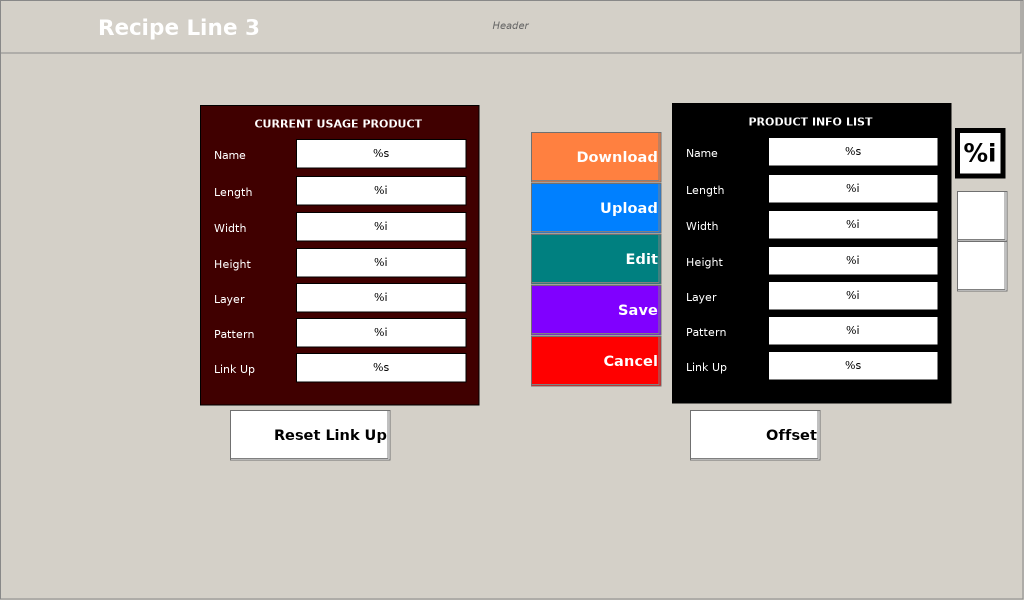
VISUALIZATION MRecipe_3  // 1024x600
    Frame (0,-2 1021x55)
        shows Header()
    Label (95,15 250x25), "Recipe Line 3"
    RoundedRectangle (672,103 279x300)
    Label (697,102 227x40), "PRODUCT INFO LIST"
    Label (683,136 78x35), "Name"
    RoundedRectangle (768,137 170x29), "%s", text variable: HMI_GVL.arRecipeHMI[3].ProductName, input disabled if: Status_GVL.StsEdit[3]
        OnMouseClick: write the text variable via Default
    Label (683,173 78x35), "Length"
    RoundedRectangle (768,174 170x29), "%i", text variable: HMI_GVL.arRecipeHMI[3].ProductLength, input disabled if: Status_GVL.StsEdit[3]
        OnMouseClick: write the text variable via Default
    Label (683,209 78x35), "Width"
    RoundedRectangle (768,210 170x29), "%i", text variable: HMI_GVL.arRecipeHMI[3].ProductWidth, input disabled if: Status_GVL.StsEdit[3]
        OnMouseClick: write the text variable via Default
    Label (683,245 78x35), "Height"
    RoundedRectangle (768,246 170x29), "%i", text variable: HMI_GVL.arRecipeHMI[3].ProductHeight, input disabled if: Status_GVL.StsEdit[3]
        OnMouseClick: write the text variable via Default
    Label (683,280 78x35), "Layer"
    RoundedRectangle (768,281 170x29), "%i", text variable: HMI_GVL.arRecipeHMI[3].Stacking, input disabled if: Status_GVL.StsEdit[3]
        OnMouseClick: write the text variable via Default
    Label (683,315 78x35), "Pattern"
    RoundedRectangle (768,316 170x29), "%i", text variable: HMI_GVL.arRecipeHMI[3].ProductPattern, input disabled if: Status_GVL.StsEdit[3]
        OnMouseClick: write the text variable via Default
    Label (683,350 78x35), "Link Up"
    RoundedRectangle (768,351 170x29), "%s", text variable: HMI_GVL.arRecipeHMI[3].LinkUpSource, input disabled if: Status_GVL.StsEdit[3]
        OnMouseClick: write the text variable via Default
    Button (531,132 130x50), "Download", image: VisuSymbols.Symbols.Download
        tap Status_GVL.Download[3]
    Button (531,183 130x50), "Upload", image: VisuSymbols.Symbols.Eject
        tap Status_GVL.Upload[3]
    Button (531,234 130x50), "Edit", image: VisuSymbols.Symbols.Edit
        tap Status_GVL.Edit[3]
    Button (531,285 130x50), "Save", invisible if: Status_GVL.StsEdit[3], image: VisuSymbols.Symbols.Save
        tap Status_GVL.Save[3]
    Button (531,336 130x50), "Cancel", invisible if: Status_GVL.StsEdit[3], image: VisuSymbols.Symbols.Wrong
        tap Status_GVL.Cancel[3]
    RoundedRectangle (955,128 50x50), "%i", text variable: Status_GVL.RecipeNumber[3]
        OnMouseClick: write the text variable via Default
    Button (957,191 50x50), image: VisuSymbols.Symbols.TriangleUp
        OnMouseClick: execute {
            IF Status_GVL.StsEdit[3] THEN
            Status_GVL.RecipeNumber[3] := Status_GVL.RecipeNumber[3]+1;
            END_IF
        }
    Button (957,241 50x50), image: VisuSymbols.Symbols.TriangleDown
        OnMouseClick: execute {
            IF Status_GVL.StsEdit[3] THEN
            Status_GVL.RecipeNumber[3] := Status_GVL.RecipeNumber[3]-1;
            END_IF
        }
    Button (690,410 130x50), "Offset", image: VisuSymbols.Symbols.Centered
        OnMouseClick: OpenDialog Dialog=MOffset_3, OpenModal=True, OpenCentered=True, PositionY=0
    Group (200,104 279x356)
        RoundedRectangle (0,1 279x300)
        Label (25,0 227x40), "CURRENT USAGE PRODUCT"
        Label (11,34 78x35), "Name"
        RoundedRectangle (96,35 170x29), "%s", text variable: Status_GVL.RecipeLine[3].ProductName
        Label (11,71 78x35), "Length"
        RoundedRectangle (96,72 170x29), "%i", text variable: Status_GVL.RecipeLine[3].ProductLength
        Label (11,107 78x35), "Width"
        RoundedRectangle (96,108 170x29), "%i", text variable: Status_GVL.RecipeLine[3].ProductWidth
        Label (11,143 78x35), "Height"
        RoundedRectangle (96,144 170x29), "%i", text variable: Status_GVL.RecipeLine[3].ProductHeight
        Label (11,178 78x35), "Layer"
        RoundedRectangle (96,179 170x29), "%i", text variable: Status_GVL.RecipeLine[3].Stacking
        Label (11,213 78x35), "Pattern"
        RoundedRectangle (96,214 170x29), "%i", text variable: Status_GVL.RecipeLine[3].ProductPattern
        Label (11,248 78x35), "Link Up"
        RoundedRectangle (96,249 170x29), "%s", text variable: Status_GVL.RecipeLine[3].LinkUpSource
        Button (30,306 160x50), "Reset Link Up", image: VisuSymbols.Symbols.Eraser
            tap HMI_GVL.Reset_LinkUp[3]
END_VISUALIZATION

(* stored: Version 1.1.0.1, ProductVersion 3.1.4024.12
   Visu MRecipe_3: Id {2ccef125-6e3e-4886-9073-ec2b294d810e} *)
